TYPE E_ContactorPosition :
(
    UNDEFINED := 0,     // Belirsiz durum (ilk çalıştırma)
    OFF := 1,           // Kontaktör kapalı
    ON := 2             // Kontaktör açık
);
END_TYPE

(* stored: Version 1.1.0.1, ProductVersion 3.1.4024.15
   EnumerationTextList E_ContactorPosition: Id {cfdeab40-25d7-43cd-b380-a905bab5b3b6} *)
